//TrajectoryControl:
//GW2 side of the interface to GW3
FUNCTION_BLOCK TrajectoryControl
VAR_INPUT
	//interface to GW3
	// INPUTS to GW3
	xBoEnable AT%Q*: BOOL := FALSE;					// Freigabesignal für Fahrt, Roboter stoppt bei FALSE
	xIntMoveToEndPosition AT%Q*: INT := 0;			// Anfahrt (in Sperrzone vor Tasche oder Ladestation) = 1, Fahrt = 0
	waypointList AT%Q*: ARRAY[0..100] OF RobotPoseSimple;	// Wegpunktliste mit Roboter-Posen in globalen Koordinaten (x, y, theta)
	newWaypointListAvailable AT%Q*: BOOL := FALSE;	// Status-Bit zur Signalisierung einer neuen WP-Liste
END_VAR
VAR_OUTPUT
	// OUTPUTS from GW3
	yBoDriving AT%I*: BOOL;							// TRUE, wenn Roboter fährt				
	yBoArrivedAtDestination AT%I*:	BOOL := FALSE;	// TRUE, wenn Ziel erreicht, Ziel entspricht letzten gültigen WP
	yUintWaypointIndex AT%I*: INT := 0;			// COUNTER zur Anzeige, des Indexes des nächstes WP
	yRPposition AT%I*: RobotPoseSimple;				// aktuelle Roboterposition, für Simulationszwecke;
END_VAR

METHOD setWaypointList : BOOL
VAR_INPUT
	newWaypointList : ARRAY [0..100] OF RobotPoseSimple;
END_VAR
waypointList := newWaypointList;
END_METHOD

END_FUNCTION_BLOCK

(* stored: Version 1.1.0.1, ProductVersion 3.1.4024.11
   POU TrajectoryControl: Id {4ea89320-b636-4d60-9ddc-899c0effc681}, SpecialFunc None
   Method setWaypointList: Id {fbf19751-62c5-44dd-b948-2eb1e925692b} *)
